FUNCTION_BLOCK FB_DiagnosisTerminal
VAR_INPUT
	uiState				:REFERENCE TO UINT;
	bWcState			:REFERENCE TO BOOL;
END_VAR
VAR_OUTPUT
	bDiagnosisOK		:BOOL;
END_VAR
VAR
	bStateOK			:BOOL;
	bWcStateOK			:BOOL;		

	sTerminalState		: STRING;
	sStateStatusAll		: STRING(255);	
END_VAR

//出力する変数リセット
bDiagnosisOK:=TRUE;
bStateOK:=TRUE;
bWcStateOK:=TRUE;

IF __ISVALIDREF(uiState)=TRUE THEN
	State_Diagnosis();
	
	IF bStateOK=FALSE THEN
		bDiagnosisOK:=FALSE;
	END_IF
END_IF

IF __ISVALIDREF(bWcState)=TRUE THEN
	WcState_Diagnosis();
	
	IF bWcStateOK=FALSE THEN
		bDiagnosisOK:=FALSE;
	END_IF
END_IF

METHOD State_Diagnosis : BOOL
VAR_INPUT
END_VAR
//ターミナルのステータスをbitから診断
IF uiState.0 AND NOT uiState.1 THEN
	sTerminalState:= 'Slave in INIT state';
END_IF
IF uiState.1 AND NOT uiState.0 THEN
	sTerminalState:= 'Slave in PREOP state';
END_IF
IF uiState.0 AND uiState.1 THEN
	sTerminalState:= 'Slave in BOOTSTRAP state';
END_IF
IF uiState.2 THEN
	sTerminalState:= 'Slave in SAFEOP state';
END_IF
IF uiState.3 THEN
	sTerminalState:= 'Slave in OP state';
END_IF

//ターミナルのエラーは複数発生する可能性があるので全bitチェック
IF uiState.4 THEN
	sStateStatusAll:= 'Slave signals error. ';
ELSE
	sStateStatusAll:= '';
END_IF
IF uiState.5 THEN
	sStateStatusAll:= CONCAT( sStateStatusAll, 'Invalid vendorID. ');
ELSE
	sStateStatusAll:= CONCAT( sStateStatusAll, '');
END_IF
IF uiState.6 THEN
	sStateStatusAll:= CONCAT( sStateStatusAll, 'Initialization error occurred. ');
ELSE
	sStateStatusAll:= CONCAT( sStateStatusAll, '');
END_IF
IF uiState.7 THEN
	sStateStatusAll:= CONCAT( sStateStatusAll, 'Slave disabled. ');
ELSE
	sStateStatusAll:= CONCAT( sStateStatusAll, '');
END_IF
IF uiState.8 THEN
	sStateStatusAll:= CONCAT( sStateStatusAll, 'Slave not present. ');
ELSE
	sStateStatusAll:= CONCAT( sStateStatusAll, '');
END_IF
IF uiState.9 THEN
	sStateStatusAll:= CONCAT( sStateStatusAll, 'Slave signals link error. ');
ELSE
	sStateStatusAll:= CONCAT( sStateStatusAll, '');
END_IF
IF uiState.10 THEN
	sStateStatusAll:= CONCAT( sStateStatusAll, 'Slave signals missing link. ');
ELSE
	sStateStatusAll:= CONCAT( sStateStatusAll, '');
END_IF
IF uiState.11 THEN
	sStateStatusAll:= CONCAT( sStateStatusAll, 'Slave signals unexpected link. ');
ELSE
	sStateStatusAll:= CONCAT( sStateStatusAll, '');
END_IF
IF uiState.12 THEN
	sStateStatusAll:= CONCAT( sStateStatusAll,  'Communication port A. ');
ELSE
	sStateStatusAll:= CONCAT( sStateStatusAll, '');
END_IF
IF uiState.13 THEN
	sStateStatusAll:= CONCAT( sStateStatusAll, 'Communication port B. ');
ELSE
	sStateStatusAll:= CONCAT( sStateStatusAll, '');
END_IF
IF uiState.14 THEN
	sStateStatusAll:= CONCAT( sStateStatusAll, 'Communication port C. ');
ELSE
	sStateStatusAll:= CONCAT( sStateStatusAll, '');
END_IF
IF uiState.15 THEN
	sStateStatusAll:= CONCAT( sStateStatusAll,  'Communication port D. ');
ELSE
	sStateStatusAll:= CONCAT( sStateStatusAll, '');
END_IF

//チェック結果を返す
IF sTerminalState= 'Slave in OP state' AND  sStateStatusAll= '' THEN
	bStateOK:= TRUE;
ELSE
	bStateOK:=FALSE;
END_IF
END_METHOD

METHOD WcState_Diagnosis : BOOL
VAR_INPUT
END_VAR
//ワーキングカウンターチェック
IF bWcState = 0 THEN
	bWcStateOK:=TRUE;
ELSE
	bWcStateOK:=FALSE;
END_IF
END_METHOD

END_FUNCTION_BLOCK

(* stored: Version 1.1.0.1, ProductVersion 3.1.4024.12
   POU FB_DiagnosisTerminal: Id {91eeac0d-8ecb-4fac-ba62-a6a0c4d5b6a5}, SpecialFunc None
   Method State_Diagnosis: Id {efd7d053-6627-49c9-8500-27a3f7aecfef}
   Method WcState_Diagnosis: Id {a838fd89-d69b-4bd9-87d8-a4f23c3eb44e} *)
